{attribute 'pack_mode' = '1'}
TYPE ST_AnalogueValueWithBinaryStatus :
STRUCT
	Value : REAL;
	BinaryStatus : BOOL;
END_STRUCT
END_TYPE

(* stored: Version 1.1.0.1, ProductVersion 3.1.4024.9
   DUT ST_AnalogueValueWithBinaryStatus: Id {357285cb-bfb4-426b-a8a1-75f1333f3bb3} *)
